PROGRAM OP130_Initialization_Seq
VAR
	temp3: BOOL;
END_VAR

IF OP130_LH_HomeOK AND OP130_GVL.SR130_Stepper_Control.Axis_In_Home AND OP130_RH_HomeOK THEN
   OP130_Temp_Home_OK:=TRUE;
   OP130_HomeRunning:=FALSE;
ELSE
	OP130_Temp_Home_OK:=FALSE;	
END_IF

IF (OP130_GVL.SR130_LH_Servo_Control.Axis_In_Home AND OP130_GVL.CR130_LH_Rot_Cyl.Position1 AND SR130_Clm_Stepper.bHomeDone AND SR130_Clm_Stepper.baxis_in_home_pos) THEN
	OP130_LH_HomeOK:=TRUE;
	OP130_Homing_Seq:=0;
ELSE
	OP130_LH_HomeOK:=FALSE;
END_IF

IF (OP130_GVL.SR130_RH_Servo_Control.Axis_In_Home AND OP130_GVL.CR130_RH_Rot_Cyl.Position1) THEN
	OP130_RH_HomeOK:=TRUE;
	OP130_RH_Homing_Seq:=0;
ELSE
	OP130_RH_HomeOK:=FALSE;
END_IF
	
CASE OP130_Homing_Seq OF
	
	0: IF (OP130_Auto AND NOT OP130_HomeRunning AND  NOT OP130_ErrorActive AND  NOT OP130_AutoRunning AND NOT OP130_StepRunning AND NOT OP130_Temp_Home_OK	) THEN
		OP130_HomeRunning:=TRUE;
		OP130_Homing_Seq:=10;
        OP130_RH_Homing_Seq:=10;	
	   END_IF
	   
	   10:IF SR130_stManualModeAxis_LH_Vert_Servo.actualPosition >=61  THEN
		  OP130_Homing_Seq:=20;
	      ELSE
		   OP130_Homing_Seq:=90;
		  END_IF
	   
	   20: IF (OP130_HomeRunning AND OP130_HMI_Homing)THEN 
		    
			  SR130_LH_Servo_Control.Position :=SR130_HMI_Servo_CylWork_Position;
			  SR130_LH_Servo_Control.velocity :=SR130_HMI_Servo_CylWork_Velocity;
		      OP130_Homing_Seq:=30;
	   END_IF
	   
	   30: IF (OP130_HomeRunning AND OP130_HMI_Homing)THEN 
		    
			SR130_LH_Servo_Control.ABSmove_Start := TRUE;
			 OP130_Homing_Seq:=35;
	   END_IF
	   
	   35 : IF (OP130_HomeRunning AND OP130_HMI_Homing)THEN 
		   	   SR130_Stepper_Control.Bsethome:=1;
			   IF SR130_Stepper_Control.Axis_In_Home THEN
				  OP130_Homing_Seq:=40; 
			   END_IF
	        END_IF
	   
	   40:IF (OP130_HomeRunning AND OP130_HMI_Homing)THEN 
		   IF OP130_GVL.SR130_LH_Servo_Control.Axis_In_Pos THEN
			 SR130_LH_Servo_Control.ABSmove_Start := FALSE;
			 OP130_Homing_Seq:=50;
		   END_IF
	      END_IF
	   
	   50:IF (OP130_HomeRunning AND OP130_HMI_Homing)THEN 
		   IF CR130_LH_Rot_Cyl.Position2 THEN
			   OP130_Homing_Seq:=60; 
		  ELSE
		   OP130_GVL.CR130_LH_Rot_Cyl.HomingCmd2:= TRUE;
		   OP130_GVL.CR130_LH_Rot_Cyl.HomingCmd1:= FALSE;
	      END_IF
	      END_IF
		  
	   60:IF (OP130_HomeRunning AND OP130_HMI_Homing)THEN 
		    
			 SR130_LH_Servo_Control.Position := SR130_HMI_Servo_Rotation_Position;
			 SR130_LH_Servo_Control.Velocity := SR130_HMI_Servo_Rotation_Velocity;
		     OP130_Homing_Seq:=70;
	      END_IF
		  
	   70: IF (OP130_HomeRunning AND OP130_HMI_Homing)THEN 
		     
		      SR130_LH_Servo_Control.ABSmove_Start := TRUE;
			  OP130_Homing_Seq:=75;
			 END_IF
	   
	   75:IF  OP130_GVL.SR130_LH_Servo_Control.Axis_In_Pos THEN 
		      SR130_LH_Servo_Control.ABSmove_Start := FALSE;
              OP130_Homing_Seq:=80;
	      END_IF
	   
	   
	   80:IF (OP130_HomeRunning AND OP130_HMI_Homing)THEN 
		      IF OP130_GVL.CR130_LH_Rot_Cyl.Position1 THEN
			     OP130_Homing_Seq:=90;
			   ELSE
				OP130_GVL.CR130_LH_Rot_Cyl.HomingCmd1:= TRUE;
				OP130_GVL.CR130_LH_Rot_Cyl.HomingCmd2:= FALSE;
		       END_IF
	       END_IF
	
	   90:IF (OP130_HomeRunning AND OP130_HMI_Homing)THEN  
			   SR130_LH_Servo_Control.position := 0.0;
			   SR130_LH_Servo_Control.Velocity := 10;
		       OP130_Homing_Seq:=100;
	      END_IF
	
	100:IF (OP130_HomeRunning AND OP130_HMI_Homing)THEN 
       		
			SR130_LH_Servo_Control.ABSmove_Start := TRUE;
			OP130_Homing_Seq:=115;
			END_IF
			
	115:IF SR130_LH_Servo_Control.Axis_In_Pos THEN
		  
		   SR130_LH_Servo_Control.ABSmove_Start := FALSE;
		   SR130_Stepper_Control.Bsethome := TRUE;
			IF SR130_Clm_Stepper.bHomeDone AND SR130_Clm_Stepper.baxis_in_home_pos THEN
			    OP130_Homing_Seq:=116;
            END_IF
		END_IF
	
    116: IF OP130_LH_HomeOK AND OP130_RH_HomeOK THEN
		    OP130_Homing_Seq:=120;
	     END_IF

	120: OP130_HomeRunning:=FALSE;
		 OP130_Homing_Seq:=0;
		
	
END_CASE





IF NOT OP130_HomeRunning THEN
	
	OP130_GVL.CR130_LH_Rot_Cyl.HomingCmd1:= FALSE;
	OP130_GVL.CR130_LH_Rot_Cyl.HomingCmd2:= FALSE;
	OP130_GVL.CR130_RH_Rot_Cyl.HomingCmd1:= FALSE;
	OP130_GVL.CR130_RH_Rot_Cyl.HomingCmd2:= FALSE;
				
END_IF

END_PROGRAM

(* stored: Version 1.1.0.1, ProductVersion 3.1.4024.11
   POU OP130_Initialization_Seq: Id {cf9366a5-5ec2-4a47-b647-2f5bb5c2020d}, SpecialFunc None *)
